// TIA Portal V18 export
FUNCTION_BLOCK "BRK_FB"   // FB21, FBD
{ S7_Optimized_Access := 'TRUE' }
VERSION : 0.1
// stored: AutoNumber true, IsIECCheckEnabled false, IsRetainMemResEnabled false, MemoryReserve 100, SetENOAutomatically false, UDAEnableTagReadback false
   VAR_INPUT
      SpeedZero : Bool;
      fwd : Bool;
      rev : Bool;
      pt : Time := T#100ms;
      error : Bool;
   END_VAR
   VAR_OUTPUT
      BRK_REL { ExternalAccessible := 'False'; ExternalVisible := 'False'; ExternalWritable := 'False'} : Bool;
   END_VAR
   VAR
      IEC_Timer_0_Instance { S7_SetPoint := 'True'} : TOF_TIME;
   END_VAR
BEGIN

REGION Network 2
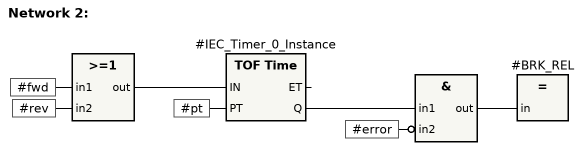
   #IEC_Timer_0_Instance(IN := #fwd OR #rev, PT := #pt);   // TOF
   #BRK_REL := #IEC_Timer_0_Instance.Q AND NOT #error;
END_REGION
END_FUNCTION_BLOCK
